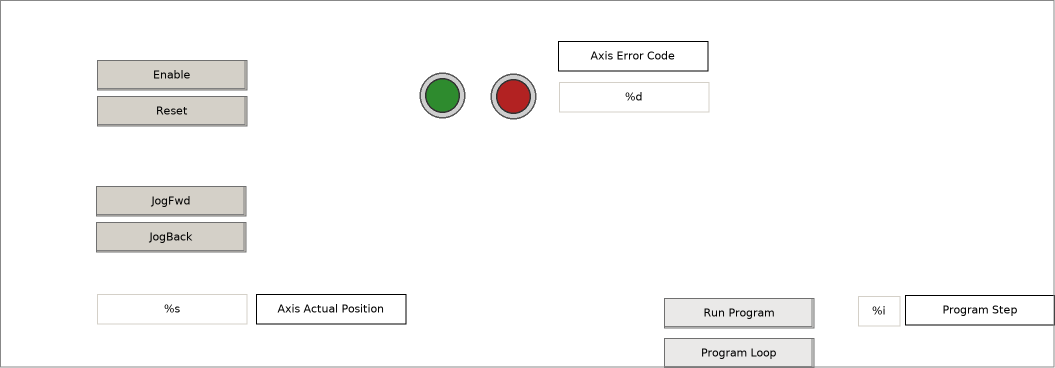
VISUALIZATION VisualizationTwinCAT  // 1055x368
    Button (96,186 150x30), "JogFwd"
        OnMouseDown: toggle MAIN.bJogForward
        OnMouseUp: toggle MAIN.bJogForward
    Button (96,222 150x30), "JogBack"
        OnMouseDown: toggle MAIN.bJogBackward
        OnMouseUp: toggle MAIN.bJogBackward
    Lamp1 (416,67 53x57), variable: MAIN.Axis1.Status.Operational, style: Lamp-Lamp1-Green
    Lamp1 (487,69 53x55), variable: MAIN.bError, style: Lamp-Lamp1-Red
    Button (97,60 150x30), "Enable"
        OnMouseDown: toggle MAIN.bJogEnable
    Button (97,96 150x30), "Reset"
        OnMouseDown: toggle MAIN.bJogReset
        OnMouseUp: toggle MAIN.bJogReset
    Textfield (559,82 150x30), "%d", text variable: MAIN.DriveErrorCode
    Textfield (97,294 150x30), "%s", text variable: MAIN.Axis1.NcToPlc.ActPos
    Button (664,298 150x30), "Run Program", colour toggle: MAIN.StartSeq
        OnMouseDown: toggle MAIN.StartSeq
    Textfield (858,296 42x30), "%i", text variable: MAIN.Sequence.i
    Rectangle (558,41 150x30), "Axis Error Code"
    Rectangle (256,294 150x30), "Axis Actual Position"
    Rectangle (905,295 150x30), "Program Step"
    Button (664,338 150x30), "Program Loop", colour toggle: MAIN.bRunContinuous, invisible if: NOT MAIN.StartSeq
        OnMouseDown: toggle MAIN.bRunContinuous
END_VISUALIZATION

(* stored: Version 1.1.0.1, ProductVersion 3.1.4024.12
   Visu VisualizationTwinCAT: Id {6686dede-6907-4126-a512-2ecbaaa45569} *)
